	DATA_BLOCK DB116
	TITLE =DBG016M  CCOMPRESSED AIR PRESSURE STEEP 5 - 8
	//COPYRIGHT:    (C) 2009  BUHLER AG, CH-9240 UZWIL, SWITZERLAND
	//
	//PRODUCT:      WinCoS_BIW01_09
	//
	//TITLE:        CCOMPRESSED AIR PRESSURE STEEP 5 - 8
	//                Machine group DB
	//                Maschinengruppen-DB
	//
	//-------------------------------------------------------------------------
	//
	//IDENT:        AUTHOR:             DEPT:             DATE:
	//
	//P01_DB116.1.0 K.Renz              CSB41             13.Jan.2010
	//              1st Release
	//
	//-------------------------------------------------------------------------
	//
	//PURPOSE:
	//
	//MANUAL :
	//
	//RESTRICTIONS:
	//
	//-------------------------------------------------------------------------
	AUTHOR  : KR
	FAMILY  : USW
	NAME    : DBG016M
	VERSION : 00.00

	FB116
	BEGIN
	      #Gr.Par.ParObjectNo 	:=1600;
	      #Gr.Par.ParIdling      	:=30;
	      #Gr.Par.ParMgr	        :=True;
	      #Gr.Par.ParWgr	        :=False;
	      #Gr.Par.ParGgr	        :=False;
	      #Gr.Par.ParEmptyingTime 	:=0;
	      #Gr.Par.ParHornCode       :=1;
	//Parameter =A-1152-MXZ11 : COMPRESSED AIR ST 5 - 8
	      #A_1152_MXZ11.Par.ParObjectNo                             :=1601;
	      #A_1152_MXZ11.Par.ParMsgType                              :=7053;
	      #A_1152_MXZ11.Par.ParHornCode                             :=1;
	      #A_1152_MXZ11.Par.ParMonTime                              :=20;
	      #A_1152_MXZ11.Par.ParStartingTime                         :=20;
	      #A_1152_MXZ11.Par.ParStoppingTime                         :=0;
	      #A_1152_MXZ11.Par.ParIdlingTime                           :=0;
	      #A_1152_MXZ11.Par.ParDelayTime                            :=10;
	      #A_1152_MXZ11.Par.ParLogOff                               :=False;
	      #A_1152_MXZ11.Par.ParManual                               :=True;
	      #A_1152_MXZ11.Par.ParRestartDelay                         :=False;
	      #A_1152_MXZ11.Par.Par2Speed                               :=False;
	      #A_1152_MXZ11.Par.ParHeavyStartup                         :=False;
	//
	//
	END_DATA_BLOCK
